
FUNCTION CB_sint_to_dword : DWORD

TITLE = ' Convert an integer into a Dword '
VERSION : '1.0'
AUTHOR  : CB
NAME    : sinToDwo
FAMILY  : TNI

VAR_INPUT
    IN : INT;
END_VAR

BEGIN

CB_sint_to_dword := BYTE_TO_DWORD(INT_TO_BYTE(IN));

END_FUNCTION
